// TIA Portal V19 export
TYPE "LEXCHANGETRAY_typeSr1000ProfinetTelegram_busyStatusBits"
// stored: Access Published
   STRUCT
      statusByte : Byte;
      busy : Bool;
      trgBusy : Bool;
      lockBusy : Bool;
      modeBusy : Bool;
      errBusy : Bool;
      fileBusy : Bool;
   END_STRUCT;
END_TYPE
